PROGRAM S1_01_Motion_7
VAR
	HMI_Motion: FB_HMI_Control;
	Motion: FB_Motion2way;

	tMessageOffset: UINT;
	tNumMessagesPerRow: UINT;
	
	
	MyAdvanceInterlock: BOOL;
	MyReturnInterlock: BOOL;
	
	MyAutoAdvanceCondition: BOOL;
	MyAutoReturnCondition: BOOL;
	testword: WORD;
	myAdvancePrompt: BOOL;
	myReturnPrompt: BOOL;
	advancedSensor: BOOL;
	returnedSensor: BOOL;
	AdvanceCoil: BOOL;
	ReturnCoil: BOOL;
	tWaitMsgXICAdv: BOOL;
	tWaitMsgXICRet: BOOL;
	FB_SimMotion: FB_SimMotion;
	tResetDepth: BOOL;
END_VAR
VAR // added by the converter: edge detectors and wires of the graphical bodies
    _rt1 : R_TRIG;
END_VAR

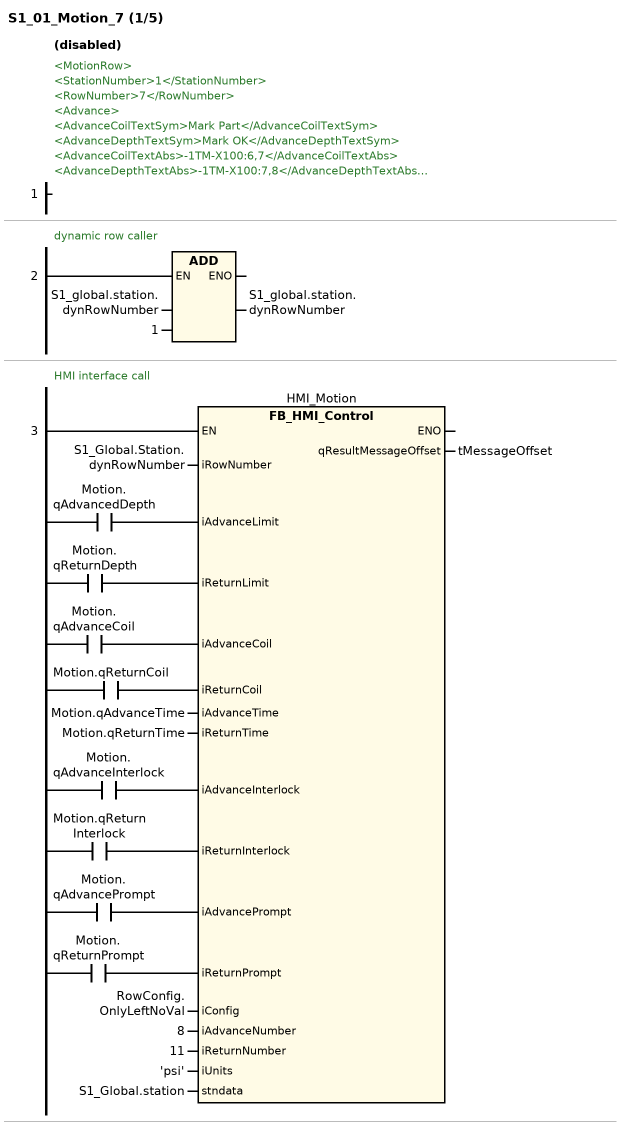
// NETWORK 1 (disabled)
// <MotionRow>
// <StationNumber>1</StationNumber>
// <RowNumber>7</RowNumber>
//   <Advance>
//     <AdvanceCoilTextSym>Mark Part</AdvanceCoilTextSym>
//     <AdvanceDepthTextSym>Mark OK</AdvanceDepthTextSym>
//     <AdvanceCoilTextAbs>-1TM-X100:6,7</AdvanceCoilTextAbs>
//     <AdvanceDepthTextAbs>-1TM-X100:7,8</AdvanceDepthTextAbs>
//     <ManSeq>8</ManSeq>
//   </Advance>
//   <Return>
//     <ReturnCoilTextSym>Return</ReturnCoilTextSym>
//     <ReturnDepthTextSym>Returned</ReturnDepthTextSym>
//     <ReturnCoilTextAbs>Q1.1</ReturnCoilTextAbs>
//     <ReturnDepthTextAbs>I1.1</ReturnDepthTextAbs>
//    <ManSeq>2</ManSeq>
//   </Return>
//   <Motion>
//     <NameSym>Marker</NameSym>
//     <NameAbs>-1TM</NameAbs>
//   </Motion>
// </MotionRow>

// NETWORK 2
// dynamic row caller
S1_global.station.dynRowNumber := S1_global.station.dynRowNumber + 1;

// NETWORK 3
// HMI interface call
HMI_Motion(
    iRowNumber := S1_Global.Station.dynRowNumber,
    iAdvanceLimit := Motion.qAdvancedDepth,
    iReturnLimit := Motion.qReturnDepth,
    iAdvanceCoil := Motion.qAdvanceCoil,
    iReturnCoil := Motion.qReturnCoil,
    iAdvanceTime := Motion.qAdvanceTime,
    iReturnTime := Motion.qReturnTime,
    iAdvanceInterlock := Motion.qAdvanceInterlock,
    iReturnInterlock := Motion.qReturnInterlock,
    iAdvancePrompt := Motion.qAdvancePrompt,
    iReturnPrompt := Motion.qReturnPrompt,
    iConfig := RowConfig.OnlyLeftNoVal,
    iAdvanceNumber := 8,
    iReturnNumber := 11,
    iUnits := 'psi',
    stndata := S1_Global.station,
    qResultMessageOffset => tMessageOffset); // FB_HMI_Control

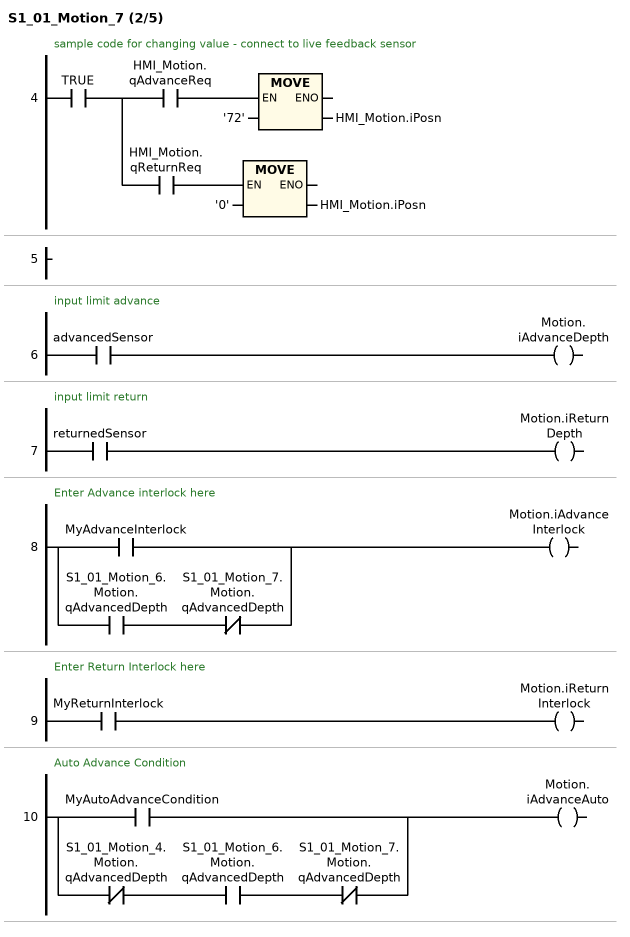
// NETWORK 4
// sample code for changing value - connect to live feedback sensor
IF TRUE AND HMI_Motion.qAdvanceReq THEN HMI_Motion.iPosn := '72'; END_IF
IF TRUE AND HMI_Motion.qReturnReq THEN HMI_Motion.iPosn := '0'; END_IF

// NETWORK 5

// NETWORK 6
// input limit advance
Motion.iAdvanceDepth := advancedSensor;

// NETWORK 7
// input limit return
Motion.iReturnDepth := returnedSensor;

// NETWORK 8
// Enter Advance interlock here
Motion.iAdvanceInterlock := MyAdvanceInterlock OR S1_01_Motion_6.Motion.qAdvancedDepth AND NOT S1_01_Motion_7.Motion.qAdvancedDepth;

// NETWORK 9
// Enter Return Interlock here
Motion.iReturnInterlock := MyReturnInterlock;

// NETWORK 10
// Auto Advance Condition
Motion.iAdvanceAuto := MyAutoAdvanceCondition OR NOT S1_01_Motion_4.Motion.qAdvancedDepth AND S1_01_Motion_6.Motion.qAdvancedDepth AND NOT S1_01_Motion_7.Motion.qAdvancedDepth;

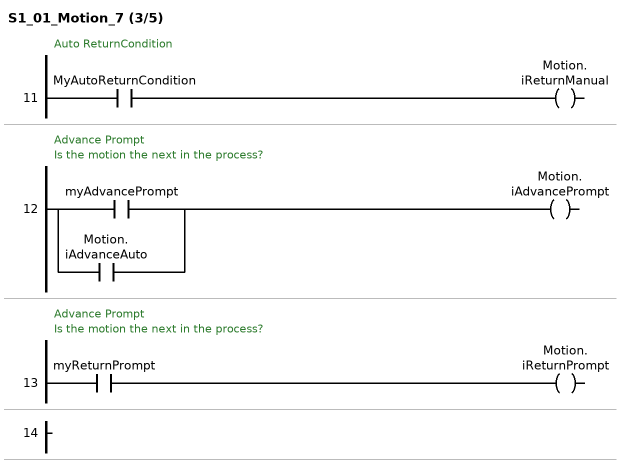
// NETWORK 11
// Auto ReturnCondition
Motion.iReturnManual := MyAutoReturnCondition;

// NETWORK 12
// Advance Prompt
// Is the motion the next in the process?
Motion.iAdvancePrompt := myAdvancePrompt OR Motion.iAdvanceAuto;

// NETWORK 13
// Advance Prompt
// Is the motion the next in the process?
Motion.iReturnPrompt := myReturnPrompt;

// NETWORK 14

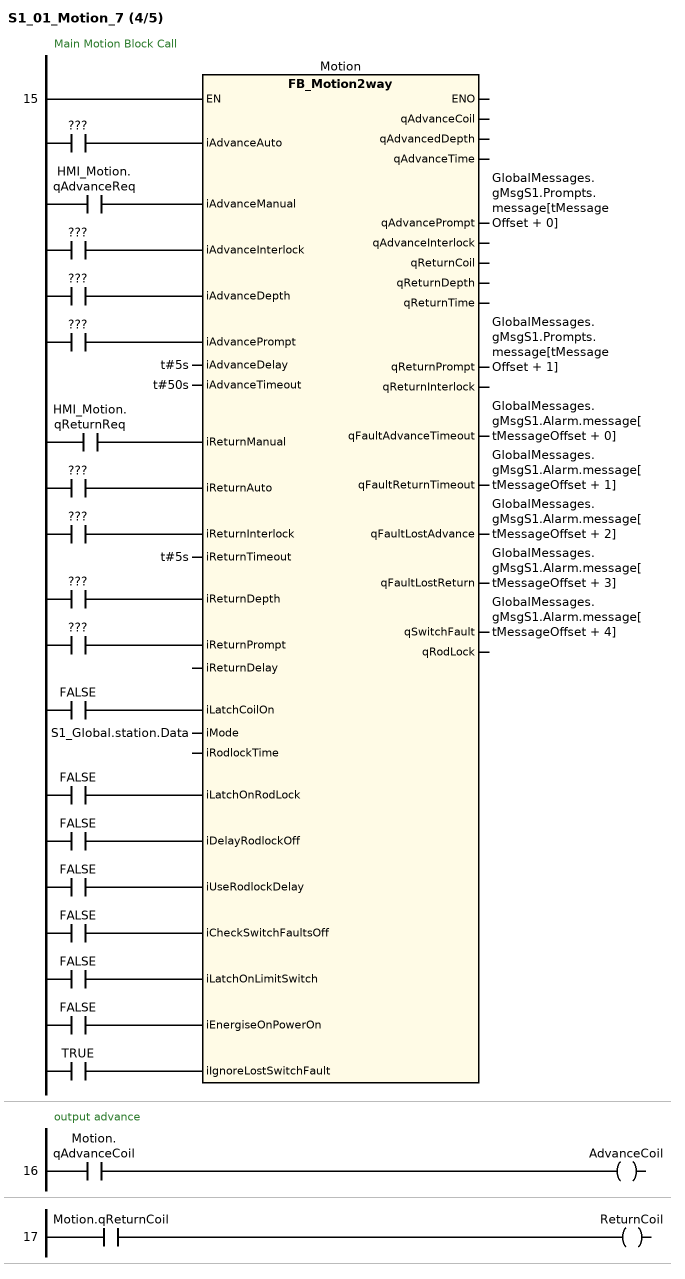
// NETWORK 15
// Main Motion Block Call
Motion(
    iAdvanceManual := HMI_Motion.qAdvanceReq,
    iAdvanceDelay := t#5s,
    iAdvanceTimeout := t#50s,
    iReturnManual := HMI_Motion.qReturnReq,
    iReturnTimeout := t#5s,
    iLatchCoilOn := FALSE,
    iMode := S1_Global.station.Data,
    iLatchOnRodLock := FALSE,
    iDelayRodlockOff := FALSE,
    iUseRodlockDelay := FALSE,
    iCheckSwitchFaultsOff := FALSE,
    iLatchOnLimitSwitch := FALSE,
    iEnergiseOnPowerOn := FALSE,
    iIgnoreLostSwitchFault := TRUE,
    qAdvancePrompt => GlobalMessages.gMsgS1.Prompts.message[tMessageOffset + 0],
    qReturnPrompt => GlobalMessages.gMsgS1.Prompts.message[tMessageOffset + 1],
    qFaultAdvanceTimeout => GlobalMessages.gMsgS1.Alarm.message[tMessageOffset + 0],
    qFaultReturnTimeout => GlobalMessages.gMsgS1.Alarm.message[tMessageOffset + 1],
    qFaultLostAdvance => GlobalMessages.gMsgS1.Alarm.message[tMessageOffset + 2],
    qFaultLostReturn => GlobalMessages.gMsgS1.Alarm.message[tMessageOffset + 3],
    qSwitchFault => GlobalMessages.gMsgS1.Alarm.message[tMessageOffset + 4]); // FB_Motion2way

// NETWORK 16
// output advance
AdvanceCoil := Motion.qAdvanceCoil;

// NETWORK 17
ReturnCoil := Motion.qReturnCoil;

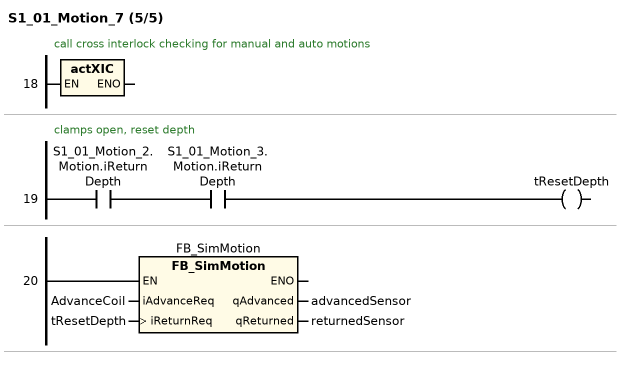
// NETWORK 18
// call cross interlock checking for manual and auto motions
actXIC();

// NETWORK 19
// clamps open, reset depth
tResetDepth := S1_01_Motion_2.Motion.iReturnDepth AND S1_01_Motion_3.Motion.iReturnDepth;

// NETWORK 20
_rt1(CLK := tResetDepth);
FB_SimMotion(
    iAdvanceReq := AdvanceCoil,
    iReturnReq := _rt1.Q,
    qAdvanced => advancedSensor,
    qReturned => returnedSensor);

ACTION actXIC:
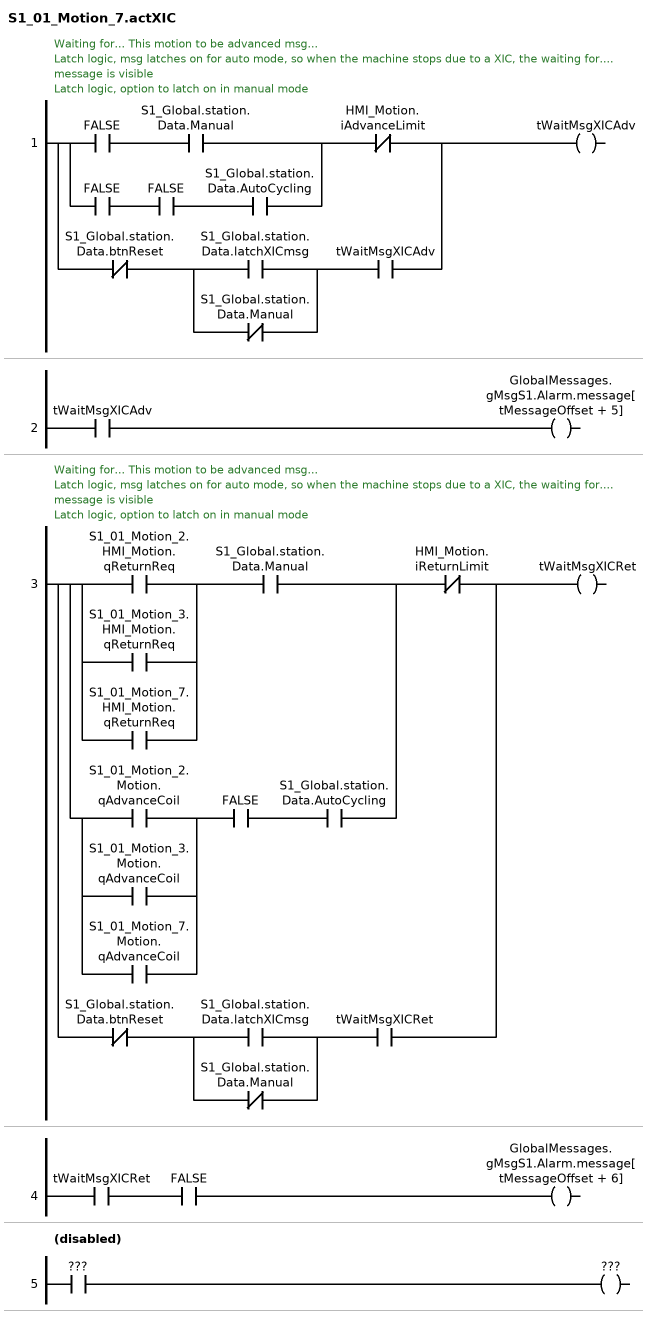
// NETWORK 1
// Waiting for... This motion to be advanced msg...
// Latch logic, msg latches on for auto mode, so when the machine stops due to a XIC, the waiting for.... message is visible
// Latch logic, option to latch on in manual mode
tWaitMsgXICAdv := (FALSE AND S1_Global.station.Data.Manual OR FALSE AND FALSE AND S1_Global.station.Data.AutoCycling) AND NOT HMI_Motion.iAdvanceLimit OR NOT S1_Global.station.Data.btnReset AND (S1_Global.station.Data.latchXICmsg OR NOT S1_Global.station.Data.Manual) AND tWaitMsgXICAdv;

// NETWORK 2
GlobalMessages.gMsgS1.Alarm.message[tMessageOffset + 5] := tWaitMsgXICAdv;

// NETWORK 3
// Waiting for... This motion to be advanced msg...
// Latch logic, msg latches on for auto mode, so when the machine stops due to a XIC, the waiting for.... message is visible
// Latch logic, option to latch on in manual mode
tWaitMsgXICRet := ((S1_01_Motion_2.HMI_Motion.qReturnReq OR S1_01_Motion_3.HMI_Motion.qReturnReq OR S1_01_Motion_7.HMI_Motion.qReturnReq) AND S1_Global.station.Data.Manual OR (S1_01_Motion_2.Motion.qAdvanceCoil OR S1_01_Motion_3.Motion.qAdvanceCoil OR S1_01_Motion_7.Motion.qAdvanceCoil) AND FALSE AND S1_Global.station.Data.AutoCycling) AND NOT HMI_Motion.iReturnLimit OR NOT S1_Global.station.Data.btnReset AND (S1_Global.station.Data.latchXICmsg OR NOT S1_Global.station.Data.Manual) AND tWaitMsgXICRet;

// NETWORK 4
GlobalMessages.gMsgS1.Alarm.message[tMessageOffset + 6] := tWaitMsgXICRet AND FALSE;

// NETWORK 5 (disabled)
// ??? := ???;
END_ACTION

END_PROGRAM

(* stored: Version 1.1.0.1, ProductVersion 3.1.4024.11
   POU S1_01_Motion_7: Id {3fb8eeb0-f560-4b3f-a64d-217de728f2b9}, SpecialFunc None
   Action actXIC: Id {cea0208b-eb1a-0abd-19b4-62b0e9c3bde7} *)
